FUNCTION_BLOCK ATM_SERVER_0_1 (* Receive a TIME as a remote OPC-UA CALL_METHOD argument via SERVER_0_1 (pairs with CLIENT_1_0/ATM_CLIENT_1_0), exposed as an ATM adapter *)
  (* Standard: 61499-2; Description: Copyright (c) 2026 HR Agrartechnik GmbH This program and the accompanying materials are made available under the terms of the Eclipse Public License 2.0 which is available at https://www.eclipse.org/legal/epl-2.0/ SPDX-License-Identifier: EPL-2.0 *)
  (* Version 1.0, 2026-09-23, Franz Höpfinger, HR Agrartechnik GmbH, initial implementation - Empfangs-Gegenstueck zu ATM_CLIENT_1_0, analog AR_SERVER_0_1/AX_SERVER_0_1 (dort REAL/BOOL statt TIME). Vorsorglich angelegt (Franz: 'die bauen wir jetzt, ich habe keinen Bock dauernd neue Runtimes zu machen'), noch kein aktueller Aufrufer. RSP wird sofort auf IND zurueckverdrahtet (SERVER_0_RSP_LATENZ-Bug, siehe Ventilsteuerung/OPC_UA_VERNETZUNG.md Punkt 12, 4s Server-Lock sonst). *)
  PACKAGE adapter::net;
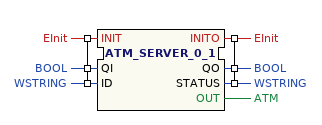
  EVENT_INPUT
    INIT : EInit WITH QI, ID; (* Initialization *)
  END_EVENT
  EVENT_OUTPUT
    INITO : EInit WITH QO, STATUS; (* Initialization Confirm *)
  END_EVENT
  VAR_INPUT
    QI : BOOL;
    ID : WSTRING;
  END_VAR
  VAR_OUTPUT
    QO : BOOL;
    STATUS : WSTRING;
  END_VAR
  PLUGS
    OUT : adapter::types::unidirectional::ATM; (* Empfangener TIME-Wert bei jedem Methodenaufruf *)
  END_PLUGS
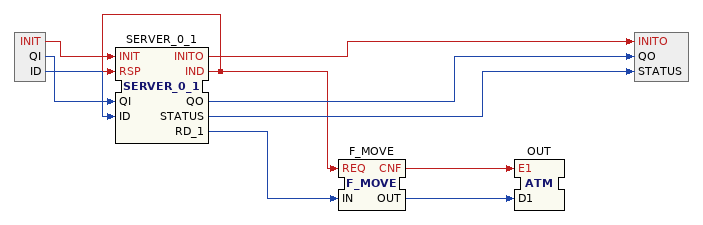
  FBS
    SERVER_0_1 : iec61499::net::SERVER_0_1;
    F_MOVE : iec61131::selection::F_MOVE; {SET_ATTRIBUTE(DataType, TIME)}
  END_FBS
  EVENT_CONNECTIONS
    INIT TO SERVER_0_1.INIT;
    SERVER_0_1.INITO TO INITO;
    SERVER_0_1.IND TO SERVER_0_1.RSP;
    SERVER_0_1.IND TO F_MOVE.REQ;
    F_MOVE.CNF TO OUT.E1;
  END_CONNECTIONS
  DATA_CONNECTIONS
    QI TO SERVER_0_1.QI;
    ID TO SERVER_0_1.ID;
    SERVER_0_1.QO TO QO;
    SERVER_0_1.STATUS TO STATUS;
    SERVER_0_1.RD_1 TO F_MOVE.IN;
    F_MOVE.OUT TO OUT.D1;
  END_CONNECTIONS
END_FUNCTION_BLOCK
